# EPICS substitutions: bcmApp/Db/bcmAmc.substitutions
########################################################################################################################
# Summary:             BCM substitutions file to generate PVs for CPSW registers
# Author:              T. Eriksen <taine@slac.stanford.edu>
# Date:                17-may-2021
# YAML config version:
########################################################################################################################

########################################################################################################################
# Macros:
#   P,R: The PV name as P:R
#   DESC, PINI, SCAN, NELM, etc.: The same fields on the records
#   PORT: The asyn port name. It must match the port name given when calling "YCPSWASYNConfig" on st.cmd
#   PARAM: The asyn paramter name. It must be defined in the dictionary file and assigned to a register
#   AMC: The AMC hardware slot (0 or 1)
########################################################################################################################

#======================================
# Register with ScalVal interfaces
#======================================

file "RegisterOut.template" { pattern
{ P,        R,              DESC,                                       PINI,   SCAN,       PORT,  PARAM       }
{ $(P), Mode,           "BCM mode"                                "NO",   "Passive",  $(PORT),    AMC$(AMC):Mode }
}

file "RegisterOutRBV.template" { pattern
{ P,           R,                DESC,                                     PINI,   SCAN,        PORT,  PARAM       }
{ $(P), ModeRBV,           "BCM mode"                                "YES",  "1 second",  $(PORT),    AMC$(AMC):Mode }
}

#======================================
# Registers with ScalVal_RO interfaces
#======================================
# Single register
file "RegisterIn.template" { pattern
{ P,          R,              DESC,                      PINI,   SCAN,       PORT,      EGU,  PARAM                  }
{ $(P), AmcClkFreq,     "AMC Clock frequency",          "YES",  "1 second", $(PORT),   "Hz", AMC$(AMC):AmcClkFreq    }
{ $(P), MuxTrigCnt,     "Valid DAQ triggers",           "YES",  "1 second", $(PORT),   "",   AMC$(AMC):MuxTrigCnt    }
{ $(P), MuxFrzStat,     "Freeze buf status",            "YES",  "1 second", $(PORT),   "",   AMC$(AMC):MuxFrzStat    }
{ $(P), MuxCascStat,    "Cascade trigger status",       "YES",  "1 second", $(PORT),   "",   AMC$(AMC):MuxCascStat   }
{ $(P), MuxTrigHwArm,   "HW trigger armed status",      "YES",  "1 second", $(PORT),   "",   AMC$(AMC):MuxTrigHwArm  }
{ $(P), MuxTrigHwStat,  "HW trigger status",            "YES",  "1 second", $(PORT),   "",   AMC$(AMC):MuxTrigHwStat }
{ $(P), MuxTrigStat,    "Combined trigger status",      "YES",  "1 second", $(PORT),   "",   AMC$(AMC):MuxTrigStat   }
{ $(P), MuxTrigSwStat,  "SW trigger status",            "YES",  "1 second", $(PORT),   "",   AMC$(AMC):MuxTrigSwStat }
{ $(P), DSPVers,        "System generator core vers",   "YES",  "1 second", $(PORT),   "",   AMC$(AMC):DSPVers       }
{ $(P), RATE,           "Trigger rate over 1 sec",      "YES",  "1 second", $(PORT),   "Hz", AMC$(AMC):RATE          }
}

# Array of register
file "RegisterArrayIn.template" { pattern
{ P,          R,             DESC,                          NELM,   PINI,   SCAN,   PORT,           PARAM           }
{ $(P), AdcData,       "Raw ADC reading",               1,     "YES",   "1 second", $(PORT),    AMC$(AMC):AdcData     }
{ $(P), MuxInDatVal,   "Incoming data valid",         4,     "YES",   "1 second", $(PORT),    AMC$(AMC):MuxInDatVal }
{ $(P), MuxStrmEna,    "Output stream enabled",       4,     "YES",   "1 second", $(PORT),    AMC$(AMC):MuxStrmEna  }
{ $(P), MuxStrmErr,    "Error during last acq",       4,     "YES",   "1 second", $(PORT),    AMC$(AMC):MuxStrmErr  }
{ $(P), MuxStrmOflw,   "Raw diag stream ctrl oflw",   4,     "YES",   "1 second", $(PORT),    AMC$(AMC):MuxStrmOflw }
{ $(P), MuxStrmPs,     "Raw diag stream ctrl pause",  4,     "YES",   "1 second", $(PORT),    AMC$(AMC):MuxStrmPs   }
{ $(P), MuxStrmRdy,    "Raw diag stream ctrl ready",  4,     "YES",   "1 second", $(PORT),    AMC$(AMC):MuxStrmRdy  }
{ $(P), MuxFrameCnt,   "4096 byte frames sent",       4,     "YES",   "1 second", $(PORT),    AMC$(AMC):MuxFrameCnt }
{ $(P), MuxTmstmp,     "Timestamp 63:0",              2,     "YES",   "1 second", $(PORT),    AMC$(AMC):MuxTmstmp   }
}

# Array of 8-bit register as a string
file "RegisterArrayChar.template" { pattern
{ P,        R,              DESC,                           NELM,   PINI,   SCAN,       PORT,  PARAM       }
}

# ENUM register
file "RegisterEnumBIn.template" { pattern
{ P,        R,              DESC,                    PINI,   ZNAM,       ONAM,       SCAN,      PORT, PARAM     }
}

#======================================
# Register with ScalVal interfaces
#======================================

# ENUM register
file "RegisterEnumBOut.template" { pattern
{ P,        R,              DESC,        PINI   ZNAM,        ONAM,     SCAN,       PORT, PARAM     }
{ $(P), AutoRearm,   "Auto rearm", "NO",  "Disabled", "Enabled", "Passive",  $(PORT),   AMC$(AMC):AutoRearm }
}

file "RegisterEnumBOutRBV.template" { pattern
{ P,        R,              DESC,         PINI    ZNAM,        ONAM,     SCAN,        PORT, PARAM     }
{ $(P), AutoRearmRBV, "Auto rearm", "YES",  "Disabled", "Enabled", ".5 second",  $(PORT),   AMC$(AMC):AutoRearm }
}

#======================================
# Register with DoubleVal_RO interfaces
#======================================

file "RegisterDoubleInLimits.template" { pattern
{ P,        R,       HOPR,   LOPR,   LOLO,    LOW,   HIGH,   HIHI   }
}

#======================================
# Register with Command interfaces
#======================================
file "RegisterCommand.template" { pattern
{ P,            R,            DESC,                            PINI,   SCAN,       PORT,   PARAM   }
}

#======================================
# Register with Stream interfaces
#======================================

file "RegisterStream.template" {pattern
{ P,            R,          DESC,               NELM,       PINI,   PORT,   PARAM       }
{ $(P),   Stream0,    "Stream channel 0",       512,    "NO",   $(PORT),     AMC$(AMC):Stream0  }
{ $(P),   Stream1,    "Stream channel 1",       512,    "NO",   $(PORT),     AMC$(AMC):Stream1  }
}

# For Stream interfaces, an additional parameter is automatically created
# and the name is generated adding ":16" to the original parameter name
# This gives access to the same stream data, but as 16-bit words which
# is the case for ADC samples for example. Note that the NELM is 2x

file "RegisterStream16.template" {pattern
{ P,            R,          DESC,                    NELM,     PINI,  PORT,  PARAM         }
{ $(P),     Stream0_16, "Stream channel 0 (16-bit)",  1024,    "NO",  $(PORT),    AMC$(AMC):Stream0:16 }
{ $(P),     Stream1_16, "Stream channel 1 (16-bit)",  1024,    "NO",  $(PORT),    AMC$(AMC):Stream1:16 }
}

#======================================
# Register with Calc interfaces
#======================================
file "RegisterCalc.template" { pattern
{ P,          R,              DESC,                           	SCAN,		EGU,  		PARAM 				}
}
